// TwinCAT 3 PLC project RedLine
// ProgramVersion: 3.1.4023.0
// libraries:
//   Tc2_Standard, * (Beckhoff Automation GmbH)
//   Tc2_System, * (Beckhoff Automation GmbH)
//   Tc3_Module, * (Beckhoff Automation GmbH)
// project tree:
//   GVLs/ GVL.TcGVL
//   / PlcTask.TcTTO (not stored)
//   POUs/ MAIN.TcPOU
// real-time tasks:
//   TASK PlcTask: cycle T#10ms, priority 20, ADS port 350
//   TASK PlcTask1: cycle T#10ms, priority 21, ADS port 351

// ---- GVLs/GVL.TcGVL
{attribute 'qualified_only'}
VAR_GLOBAL

//Block States IO
mInSwitch : ARRAY[0..76] OF DINT;
mOutSwitch : ARRAY[0..76] OF DINT;
mInOccupancies : ARRAY[0..76] OF DINT;
mOutOccupancies : ARRAY[0..76] OF DINT;
mInSpeeds : ARRAY[0..76] OF DINT;
mOutSpeeds : ARRAY[0..76] OF DINT;
mInAuthorities : ARRAY[0..76] OF DINT;
mOutAuthorities : ARRAY[0..76] OF DINT;
mInCrossings : ARRAY[0..76] OF DINT;
mOutCrossings : ARRAY[0..76] OF DINT;
mInLeftLights : ARRAY[0..76] OF DINT;
mOutLeftLights : ARRAY[0..76] OF DINT;
mInRightLights : ARRAY[0..76] OF DINT;
mOutRightLights : ARRAY[0..76] OF DINT;
mInMaintenance : ARRAY[0..76] OF DINT;
mOutMaintenance : ARRAY[0..76] OF DINT;

END_VAR

// ---- POUs/MAIN.TcPOU
PROGRAM MAIN
VAR

inc1 : DINT := 0;
	
END_VAR


FOR inc1 := 0 TO 76 DO

	GVL.mOutOccupancies[inc1] := GVL.mInOccupancies[inc1];
	GVL.mOutSpeeds[inc1] := GVL.mInSpeeds[inc1];
	GVL.mOutAuthorities[inc1] := GVL.mInAuthorities[inc1];
	GVL.mOutMaintenance[inc1] := GVL.mInMaintenance[inc1];

END_FOR

inc1 := 0;

//This starts the main track logic section

//Crossing Logic
IF GVL.mInOccupancies[46] = 0 THEN
	GVL.mOutCrossings[46] := 1;
ELSE
	GVL.mOutCrossings[46] := 0;
END_IF

//Switch Logic
IF GVL.mInMaintenance[8] = 1 THEN
    GVL.mOutSwitch[8] := GVL.mInSwitch[8];
ELSE
    IF GVL.mInOccupancies[76] = 0 THEN
    	GVL.mOutSwitch[8] := 76;
    ELSE
		GVL.mOutSwitch[8] := 9;
	END_IF
END_IF

IF GVL.mInMaintenance[15] = 1 THEN
    GVL.mOutSwitch[15] := GVL.mInSwitch[15];
ELSE
    IF GVL.mInOccupancies[14] = 0 THEN
    FOR inc1 := 16 TO 26 DO 
        IF GVL.mInOccupancies[inc1] = 0 THEN
            GVL.mOutSwitch[15] := 1;
            Exit;
        ELSE 
            GVL.mOutSwitch[15] := 14;
        END_IF
    END_FOR
	END_IF
END_IF

IF GVL.mInMaintenance[26] = 1 THEN
    GVL.mOutSwitch[26] := GVL.mInSwitch[26];
ELSE
    IF GVL.mInOccupancies[75] = 0 THEN
    FOR inc1 := 16 TO 26 DO 
        IF GVL.mInOccupancies[inc1] = 0 THEN
            GVL.mOutSwitch[26] := 27;
            Exit;
        ELSE 
            GVL.mOutSwitch[26] := 75;
        END_IF
    END_FOR
	END_IF
END_IF

IF GVL.mInMaintenance[32] = 1 THEN
    GVL.mOutSwitch[32] := GVL.mInSwitch[32];
ELSE
    IF GVL.mInOccupancies[31] = 0 THEN
    FOR inc1 := 32 TO 37 DO 
        IF GVL.mInOccupancies[inc1] = 0 THEN
            GVL.mOutSwitch[32] := 71;
            Exit;
        ELSE 
            GVL.mOutSwitch[32] := 31;
        END_IF
    END_FOR
	END_IF
END_IF

IF GVL.mInMaintenance[37] = 1 THEN
    GVL.mOutSwitch[37] := GVL.mInSwitch[37];
ELSE
    IF GVL.mInOccupancies[70] = 0 THEN
    FOR inc1 := 32 TO 37 DO 
        IF GVL.mInOccupancies[inc1] = 0 THEN
            GVL.mOutSwitch[37] := 38;
            Exit;
        ELSE 
            GVL.mOutSwitch[37] := 70;
        END_IF
    END_FOR
	END_IF
END_IF

IF GVL.mInMaintenance[43] = 1 THEN
    GVL.mOutSwitch[43] := GVL.mInSwitch[43];
ELSE
    IF GVL.mInOccupancies[42] = 0 THEN
    FOR inc1 := 43 TO 51 DO 
        IF GVL.mInOccupancies[inc1] = 0 THEN
            GVL.mOutSwitch[43] := 66;
            Exit;
        ELSE 
            GVL.mOutSwitch[43] := 42;
        END_IF
    END_FOR
	END_IF
END_IF

IF GVL.mInMaintenance[51] = 1 THEN
    GVL.mOutSwitch[51] := GVL.mInSwitch[51];
ELSE
    IF GVL.mInOccupancies[65] = 0 THEN
    FOR inc1 := 43 TO 51 DO 
        IF GVL.mInOccupancies[inc1] = 0 THEN
            GVL.mOutSwitch[51] := 52;
            Exit;
        ELSE 
            GVL.mOutSwitch[51] := 65;
        END_IF
    END_FOR
	END_IF
END_IF

END_PROGRAM
